FUNCTION_BLOCK Item_Mockup IMPLEMENTS I_Base
VAR
	_Name : T_MaxString;
END_VAR

PROPERTY Name : T_MaxString
GET
Name := _Name;
END_GET
SET
_Name := Name;
END_SET
END_PROPERTY

END_FUNCTION_BLOCK

(* stored: Version 1.1.0.1, ProductVersion 3.1.4026.18
   POU Item_Mockup: Id {6eed378d-7c89-4b79-baa5-7ceee83fb0ef}, SpecialFunc None
   Property Name: Id {9387ce54-216c-4b79-8a58-d94d54215f16}
   Get Get: Id {6f82408c-fc01-475a-96e9-a935785d42a7}
   Set Set: Id {2ab4a342-f76f-46e7-a7cb-c7be8010fedc} *)
